Staubli VAL3: start.pgx

program start()
begin
  while true
    delay(0)
  endWhile
end
